// SIMATIC S7-200 SMART project (STEP 7-Micro/WIN SMART), CPU ST20

SYMBOL_TABLE 系统符号
Always_On        SM0.0    // 始终接通
Clock_1s         SM0.5    // 针对 1 s 的周期时间，时钟脉冲接通 0.5 s，断开 0.5 s.
END_SYMBOL_TABLE

ORGANIZATION_BLOCK MAIN:OB1
TITLE=程序注释
BEGIN
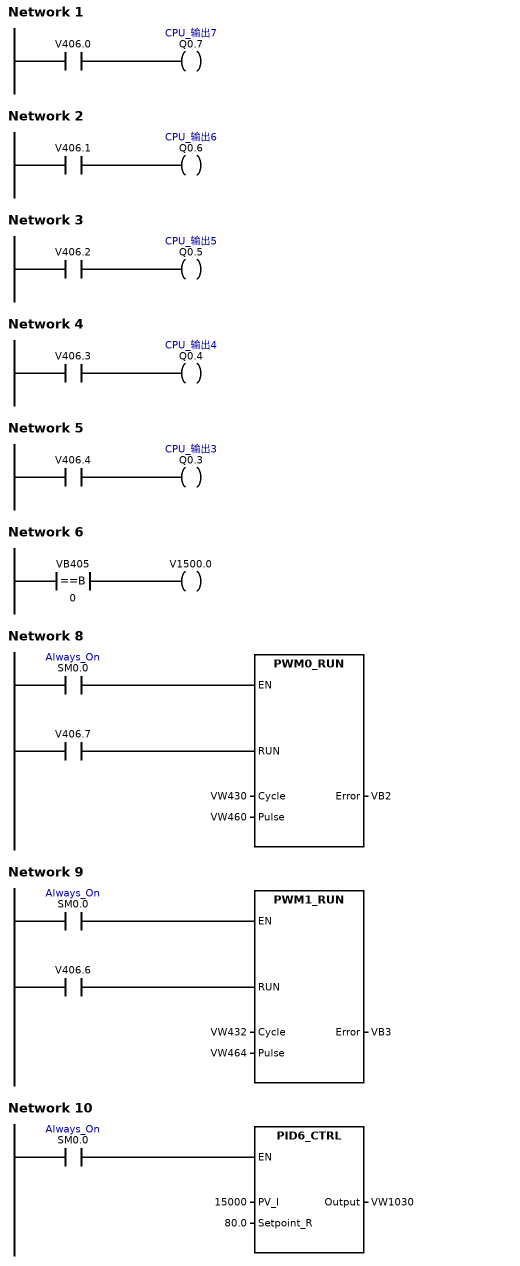
Network 1
LD     V406.0
=      CPU_输出7:Q0.7
Network 2
LD     V406.1
=      CPU_输出6:Q0.6
Network 3
LD     V406.2
=      CPU_输出5:Q0.5
Network 4
LD     V406.3
=      CPU_输出4:Q0.4
Network 5
LD     V406.4
=      CPU_输出3:Q0.3
Network 6
LDB=   VB405, 0
=      V1500.0
Network 8
LD     Always_On:SM0.0
=      L60.0
LD     V406.7
=      L63.7
LD     L60.0
CALL   PWM0_RUN:SBR3, L63.7, VW430, VW460, VB2
Network 9
LD     Always_On:SM0.0
=      L60.0
LD     V406.6
=      L63.7
LD     L60.0
CALL   PWM1_RUN:SBR4, L63.7, VW432, VW464, VB3
Network 10
LD     Always_On:SM0.0
CALL   PID6_CTRL:SBR6, 15000, 80.0, VW1030
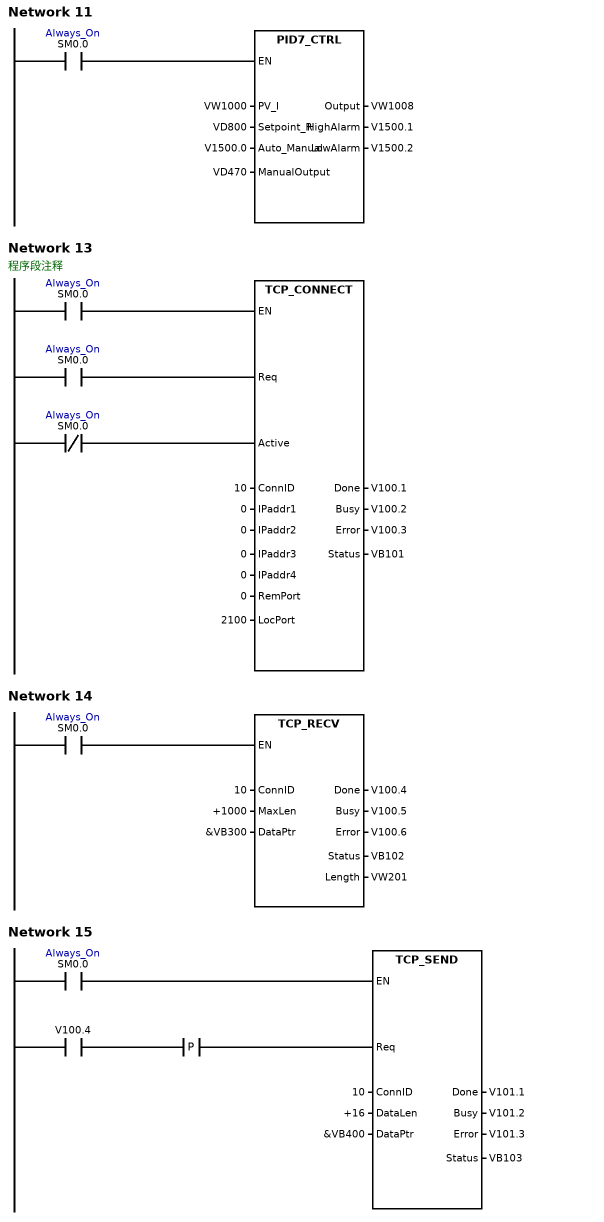
Network 11
LD     Always_On:SM0.0
CALL   PID7_CTRL:SBR7, VW1000, VD800, V1500.0, VD470, VW1008, V1500.1, V1500.2
Network 13
// 程序段注释
LD     Always_On:SM0.0
=      L60.0
LD     Always_On:SM0.0
=      L63.7
LDN    Always_On:SM0.0
=      L63.6
LD     L60.0
CALL   TCP_CONNECT:SBR1, L63.7, L63.6, 10, 0, 0, 0, 0, 0, 2100, V100.1, V100.2, V100.3, VB101
Network 14
LD     Always_On:SM0.0
CALL   TCP_RECV:SBR2, 10, +1000, &VB300, V100.4, V100.5, V100.6, VB102, VW201
Network 15
LD     Always_On:SM0.0
=      L60.0
LD     V100.4
EU
=      L63.7
LD     L60.0
CALL   TCP_SEND:SBR5, L63.7, 10, +16, &VB400, V101.1, V101.2, V101.3, VB103
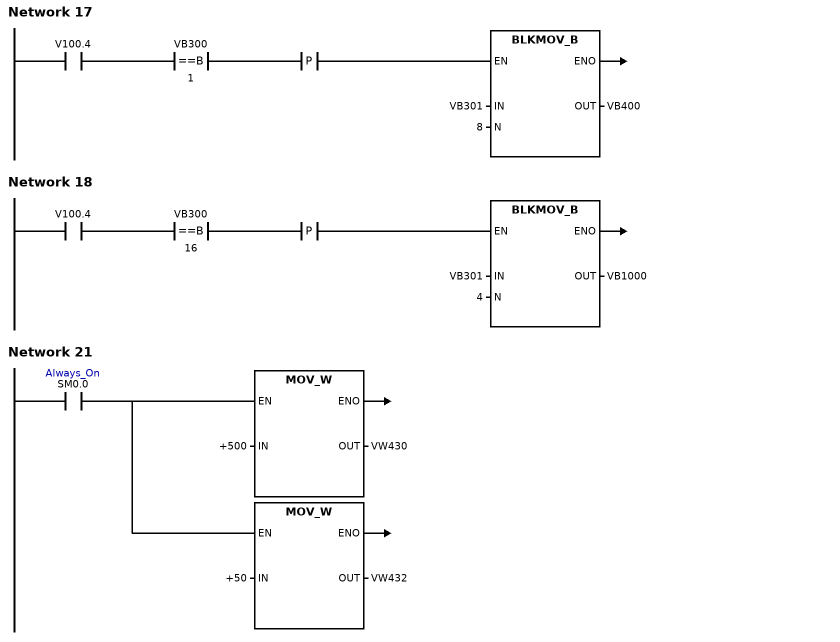
Network 17
LD     V100.4
AB=    VB300, 1
EU
BMB    VB301, VB400, 8
Network 18
LD     V100.4
AB=    VB300, 16
EU
BMB    VB301, VB1000, 4
Network 21
LD     Always_On:SM0.0
MOVW   +500, VW430
MOVW   +50, VW432
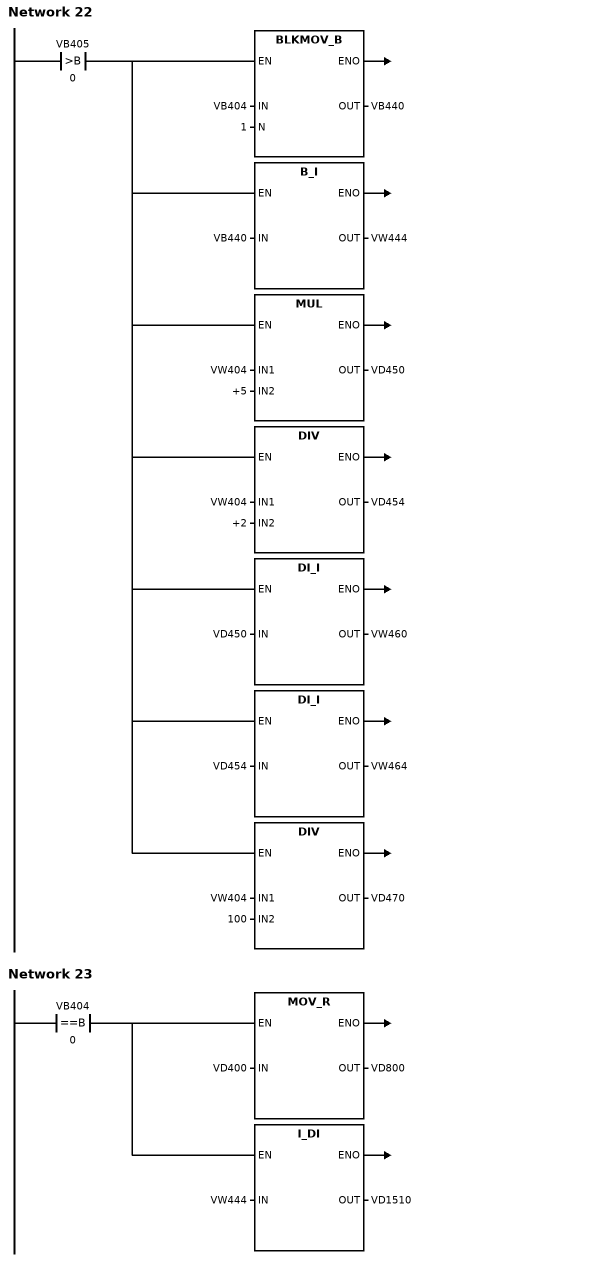
Network 22
LDB>   VB405, 0
BMB    VB404, VB440, 1
BTI    VB440, VW444
MOVW   VW404, VW452
MUL    +5, VD450
MOVW   VW404, VW456
DIV    +2, VD454
DTI    VD450, VW460
DTI    VD454, VW464
MOVW   VW404, VW472
DIV    100, VD470
Network 23
LDB=   VB404, 0
MOVR   VD400, VD800
ITD    VW444, VD1510
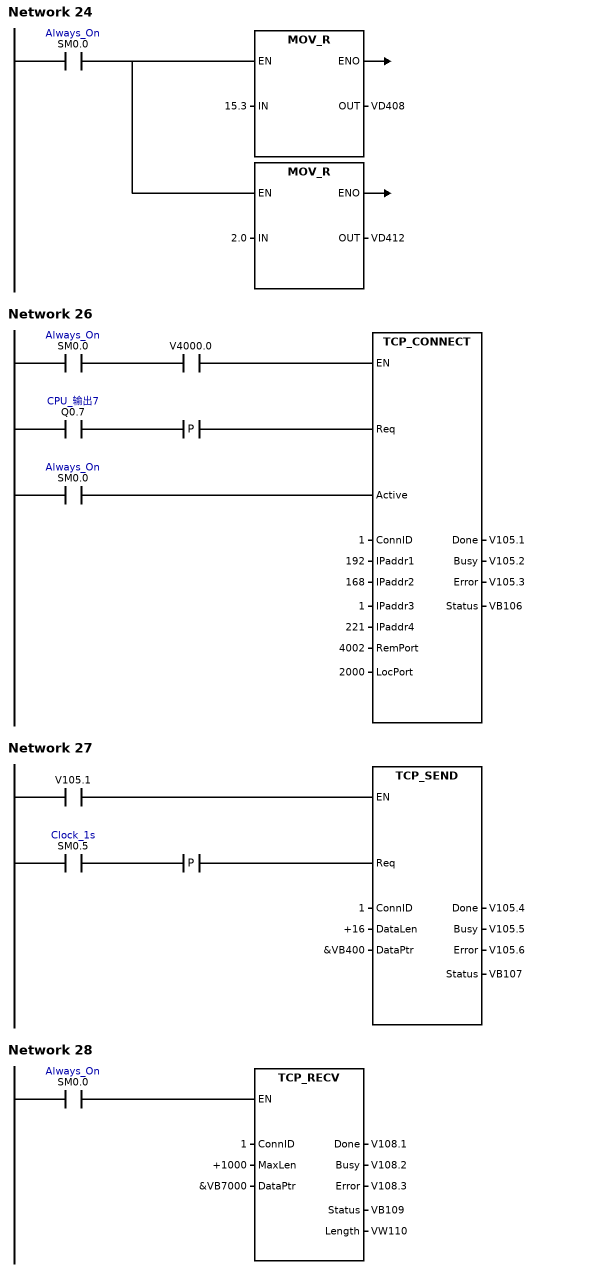
Network 24
LD     Always_On:SM0.0
MOVR   15.3, VD408
MOVR   2.0, VD412
Network 26
LD     Always_On:SM0.0
A      V4000.0
=      L60.0
LD     CPU_输出7:Q0.7
EU
=      L63.7
LD     Always_On:SM0.0
=      L63.6
LD     L60.0
CALL   TCP_CONNECT:SBR1, L63.7, L63.6, 1, 192, 168, 1, 221, 4002, 2000, V105.1, V105.2, V105.3, VB106
Network 27
LD     V105.1
=      L60.0
LD     Clock_1s:SM0.5
EU
=      L63.7
LD     L60.0
CALL   TCP_SEND:SBR5, L63.7, 1, +16, &VB400, V105.4, V105.5, V105.6, VB107
Network 28
LD     Always_On:SM0.0
CALL   TCP_RECV:SBR2, 1, +1000, &VB7000, V108.1, V108.2, V108.3, VB109, VW110
END_ORGANIZATION_BLOCK

// SBR1: protected block, not included

// SBR2: protected block, not included

// SBR3: protected block, not included

// SBR4: protected block, not included

// SBR5: protected block, not included

// SBR6: protected block, not included

// SBR7: protected block, not included

// INT1: protected block, not included
